FUNCTION_BLOCK QUARTERS_TO_BOOLS (* Composite FB wrapping other FBs *)
  (* Standard: 61499-2; Description: Copyright (c) 2024 HR Agrartechnik GmbH This program and the accompanying materials are made available under the terms of the Eclipse Public License 2.0 which is available at https://www.eclipse.org/legal/epl-2.0/ SPDX-License-Identifier: EPL-2.0 *)
  (* Version 1.0, 2024-02-29, Franz Höpfinger, HR Agrartechnik GmbH *)
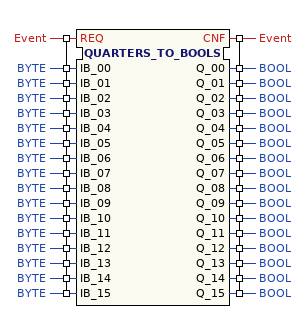
  EVENT_INPUT
    REQ WITH IB_00, IB_01, IB_02, IB_03, IB_04, IB_05, IB_06, IB_07, IB_08, IB_09, IB_10, IB_11, IB_12, IB_13, IB_14, IB_15; (* Normal Execution Request *)
  END_EVENT
  EVENT_OUTPUT
    CNF WITH Q_00, Q_01, Q_02, Q_03, Q_04, Q_05, Q_06, Q_07, Q_08, Q_09, Q_10, Q_11, Q_12, Q_13, Q_14, Q_15; (* Execution Confirmation *)
  END_EVENT
  VAR_INPUT
    IB_00 : BYTE := quarter::COMMAND_DISABLE; (* 2bit (quarter Byte) Output with 4 States *)
    IB_01 : BYTE := quarter::COMMAND_DISABLE; (* 2bit (quarter Byte) Output with 4 States *)
    IB_02 : BYTE := quarter::COMMAND_DISABLE; (* 2bit (quarter Byte) Output with 4 States *)
    IB_03 : BYTE := quarter::COMMAND_DISABLE; (* 2bit (quarter Byte) Output with 4 States *)
    IB_04 : BYTE := quarter::COMMAND_DISABLE; (* 2bit (quarter Byte) Output with 4 States *)
    IB_05 : BYTE := quarter::COMMAND_DISABLE; (* 2bit (quarter Byte) Output with 4 States *)
    IB_06 : BYTE := quarter::COMMAND_DISABLE; (* 2bit (quarter Byte) Output with 4 States *)
    IB_07 : BYTE := quarter::COMMAND_DISABLE; (* 2bit (quarter Byte) Output with 4 States *)
    IB_08 : BYTE := quarter::COMMAND_DISABLE; (* 2bit (quarter Byte) Output with 4 States *)
    IB_09 : BYTE := quarter::COMMAND_DISABLE; (* 2bit (quarter Byte) Output with 4 States *)
    IB_10 : BYTE := quarter::COMMAND_DISABLE; (* 2bit (quarter Byte) Output with 4 States *)
    IB_11 : BYTE := quarter::COMMAND_DISABLE; (* 2bit (quarter Byte) Output with 4 States *)
    IB_12 : BYTE := quarter::COMMAND_DISABLE; (* 2bit (quarter Byte) Output with 4 States *)
    IB_13 : BYTE := quarter::COMMAND_DISABLE; (* 2bit (quarter Byte) Output with 4 States *)
    IB_14 : BYTE := quarter::COMMAND_DISABLE; (* 2bit (quarter Byte) Output with 4 States *)
    IB_15 : BYTE := quarter::COMMAND_DISABLE; (* 2bit (quarter Byte) Output with 4 States *)
  END_VAR
  VAR_OUTPUT
    Q_00 : BOOL := FALSE; (* BOOL Output *)
    Q_01 : BOOL := FALSE; (* BOOL Output *)
    Q_02 : BOOL := FALSE; (* BOOL Output *)
    Q_03 : BOOL := FALSE; (* BOOL Output *)
    Q_04 : BOOL := FALSE; (* BOOL Output *)
    Q_05 : BOOL := FALSE; (* BOOL Output *)
    Q_06 : BOOL := FALSE; (* BOOL Output *)
    Q_07 : BOOL := FALSE; (* BOOL Output *)
    Q_08 : BOOL := FALSE; (* BOOL Output *)
    Q_09 : BOOL := FALSE; (* BOOL Output *)
    Q_10 : BOOL := FALSE; (* BOOL Output *)
    Q_11 : BOOL := FALSE; (* BOOL Output *)
    Q_12 : BOOL := FALSE; (* BOOL Output *)
    Q_13 : BOOL := FALSE; (* BOOL Output *)
    Q_14 : BOOL := FALSE; (* BOOL Output *)
    Q_15 : BOOL := FALSE; (* BOOL Output *)
  END_VAR
  FBS
    QUARTER_TO_BOOL_00 : QUARTER_TO_BOOL;
    QUARTER_TO_BOOL_01 : QUARTER_TO_BOOL;
    QUARTER_TO_BOOL_02 : QUARTER_TO_BOOL;
    QUARTER_TO_BOOL_03 : QUARTER_TO_BOOL;
    QUARTER_TO_BOOL_04 : QUARTER_TO_BOOL;
    QUARTER_TO_BOOL_05 : QUARTER_TO_BOOL;
    QUARTER_TO_BOOL_06 : QUARTER_TO_BOOL;
    QUARTER_TO_BOOL_07 : QUARTER_TO_BOOL;
    QUARTER_TO_BOOL_08 : QUARTER_TO_BOOL;
    QUARTER_TO_BOOL_09 : QUARTER_TO_BOOL;
    QUARTER_TO_BOOL_10 : QUARTER_TO_BOOL;
    QUARTER_TO_BOOL_11 : QUARTER_TO_BOOL;
    QUARTER_TO_BOOL_12 : QUARTER_TO_BOOL;
    QUARTER_TO_BOOL_13 : QUARTER_TO_BOOL;
    QUARTER_TO_BOOL_14 : QUARTER_TO_BOOL;
    QUARTER_TO_BOOL_15 : QUARTER_TO_BOOL;
  END_FBS
  EVENT_CONNECTIONS
    REQ TO QUARTER_TO_BOOL_00.REQ;
    QUARTER_TO_BOOL_00.CNF TO QUARTER_TO_BOOL_01.REQ;
    QUARTER_TO_BOOL_01.CNF TO QUARTER_TO_BOOL_02.REQ;
    QUARTER_TO_BOOL_03.CNF TO QUARTER_TO_BOOL_04.REQ;
    QUARTER_TO_BOOL_04.CNF TO QUARTER_TO_BOOL_05.REQ;
    QUARTER_TO_BOOL_05.CNF TO QUARTER_TO_BOOL_06.REQ;
    QUARTER_TO_BOOL_14.CNF TO QUARTER_TO_BOOL_15.REQ;
    QUARTER_TO_BOOL_15.CNF TO CNF;
    QUARTER_TO_BOOL_13.CNF TO QUARTER_TO_BOOL_14.REQ;
    QUARTER_TO_BOOL_12.CNF TO QUARTER_TO_BOOL_13.REQ;
    QUARTER_TO_BOOL_11.CNF TO QUARTER_TO_BOOL_12.REQ;
    QUARTER_TO_BOOL_10.CNF TO QUARTER_TO_BOOL_11.REQ;
    QUARTER_TO_BOOL_09.CNF TO QUARTER_TO_BOOL_10.REQ;
    QUARTER_TO_BOOL_08.CNF TO QUARTER_TO_BOOL_09.REQ;
    QUARTER_TO_BOOL_07.CNF TO QUARTER_TO_BOOL_08.REQ;
    QUARTER_TO_BOOL_06.CNF TO QUARTER_TO_BOOL_07.REQ;
    QUARTER_TO_BOOL_02.CNF TO QUARTER_TO_BOOL_03.REQ;
  END_CONNECTIONS
  DATA_CONNECTIONS
    IB_00 TO QUARTER_TO_BOOL_00.IB;
    IB_01 TO QUARTER_TO_BOOL_01.IB;
    IB_02 TO QUARTER_TO_BOOL_02.IB;
    IB_03 TO QUARTER_TO_BOOL_03.IB;
    IB_04 TO QUARTER_TO_BOOL_04.IB;
    IB_05 TO QUARTER_TO_BOOL_05.IB;
    IB_06 TO QUARTER_TO_BOOL_06.IB;
    IB_07 TO QUARTER_TO_BOOL_07.IB;
    IB_15 TO QUARTER_TO_BOOL_15.IB;
    IB_14 TO QUARTER_TO_BOOL_14.IB;
    IB_13 TO QUARTER_TO_BOOL_13.IB;
    IB_12 TO QUARTER_TO_BOOL_12.IB;
    IB_11 TO QUARTER_TO_BOOL_11.IB;
    IB_10 TO QUARTER_TO_BOOL_10.IB;
    IB_09 TO QUARTER_TO_BOOL_09.IB;
    IB_08 TO QUARTER_TO_BOOL_08.IB;
    QUARTER_TO_BOOL_15.Q TO Q_15;
    QUARTER_TO_BOOL_00.Q TO Q_00;
    QUARTER_TO_BOOL_01.Q TO Q_01;
    QUARTER_TO_BOOL_02.Q TO Q_02;
    QUARTER_TO_BOOL_03.Q TO Q_03;
    QUARTER_TO_BOOL_04.Q TO Q_04;
    QUARTER_TO_BOOL_05.Q TO Q_05;
    QUARTER_TO_BOOL_06.Q TO Q_06;
    QUARTER_TO_BOOL_07.Q TO Q_07;
    QUARTER_TO_BOOL_08.Q TO Q_08;
    QUARTER_TO_BOOL_09.Q TO Q_09;
    QUARTER_TO_BOOL_10.Q TO Q_10;
    QUARTER_TO_BOOL_11.Q TO Q_11;
    QUARTER_TO_BOOL_12.Q TO Q_12;
    QUARTER_TO_BOOL_13.Q TO Q_13;
    QUARTER_TO_BOOL_14.Q TO Q_14;
  END_CONNECTIONS
END_FUNCTION_BLOCK
